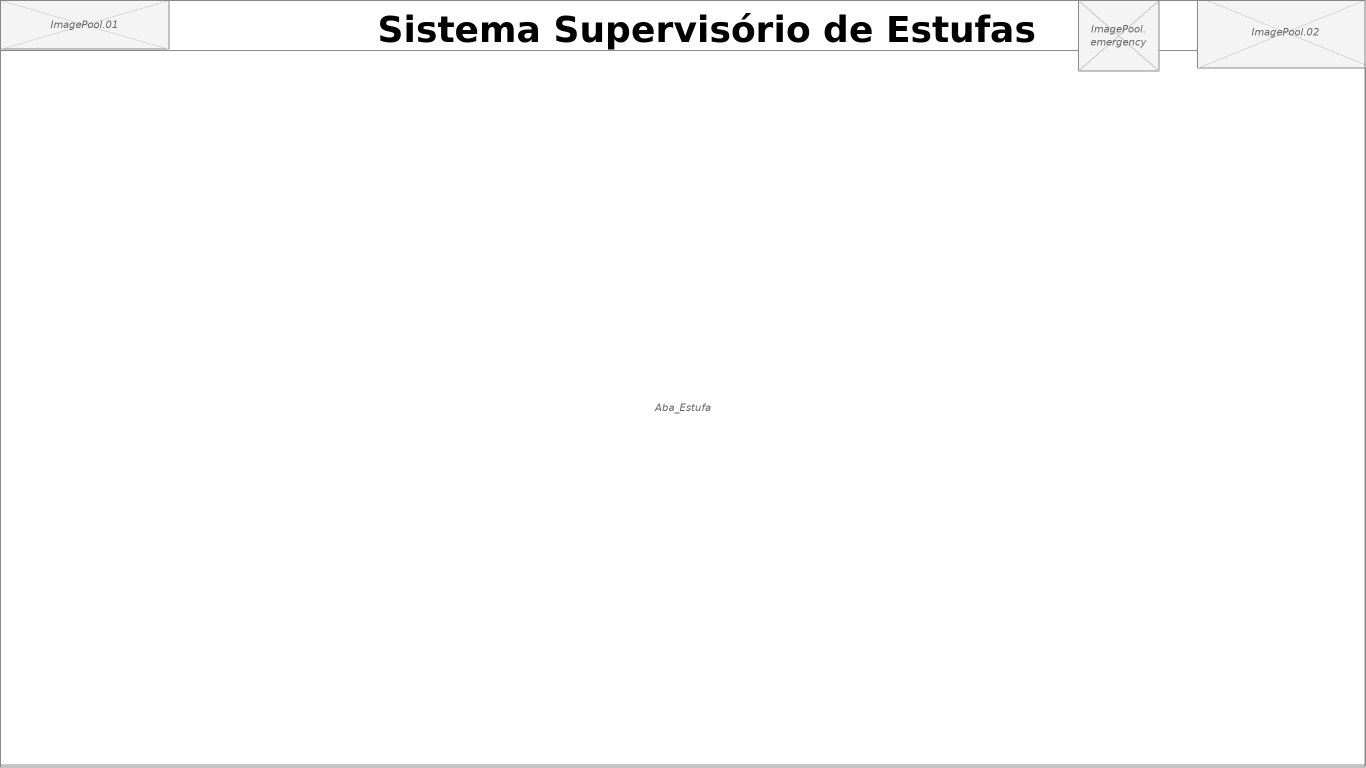
VISUALIZATION Home  // 1366x768
    TabControl (0,50 1366x715), frame switch variable: GVL.actEst
        shows Aba_Estufa()
        shows Aba_Estufa_2()
        shows Aba_Estufa_3()
        shows Aba_Manu()
        shows Historical()
        [0]: TabTitle=Estufa 203/019
        [1]: TabTitle=Estufa 203/020
        [2]: TabTitle=Estufa 203/021
        [3]: TabTitle=Manutenção
        [4]: TabTitle=Histórico
    Image (1197,-4 177x72), image: ImagePool.02
    Label (390,2 634x55), "Sistema Supervisório de Estufas"
    Image (0,0 169x49), image: ImagePool.01
    Image (1078,0 81x71), invisible if: not GVL.emergency, image: ImagePool.emergency
        OnMouseClick: execute {
            gvl.emergencia019:= FALSE;
            gvl.emergencia020:= FALSE;
            gvl.emergencia021:= FALSE;
            gvl.pwEmerg_019:= FALSE;
            gvl.pwEmerg_020:= FALSE;
            gvl.pwEmerg_021:= FALSE;
            gvl.emergency:= false;
        }
END_VISUALIZATION

(* stored: Version 1.1.0.1, ProductVersion 3.1.4024.12
   Visu Home: Id {1af690f5-949b-43d6-847b-ae8ee90bf8fd} *)
